FUNCTION_BLOCK E_SPLIT_6 (* Composite Function Block Type *)
  (* Standard: 61499-2 *)
  (* Version 0.0, 2018-11-07, 4DIAC-IDE, 4DIAC-Consortium *)
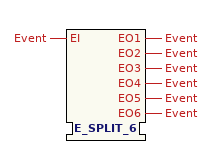
  EVENT_INPUT
    EI; (* Initialization Request *)
  END_EVENT
  EVENT_OUTPUT
    EO1; (* Initialization Confirm *)
    EO2;
    EO3;
    EO4;
    EO5;
    EO6;
  END_EVENT
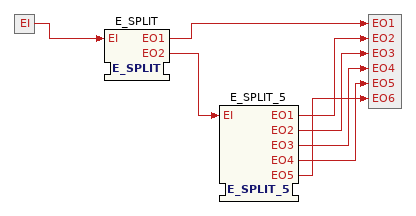
  FBS
    E_SPLIT_5 : E_SPLIT_5;
    E_SPLIT : E_SPLIT;
  END_FBS
  EVENT_CONNECTIONS
    EI TO E_SPLIT.EI;
    E_SPLIT.EO1 TO EO1;
    E_SPLIT.EO2 TO E_SPLIT_5.EI;
    E_SPLIT_5.EO1 TO EO2;
    E_SPLIT_5.EO2 TO EO3;
    E_SPLIT_5.EO3 TO EO4;
    E_SPLIT_5.EO4 TO EO5;
    E_SPLIT_5.EO5 TO EO6;
  END_CONNECTIONS
END_FUNCTION_BLOCK
